Universal Robots PolyScope program: robot_interaction_lesson.urp

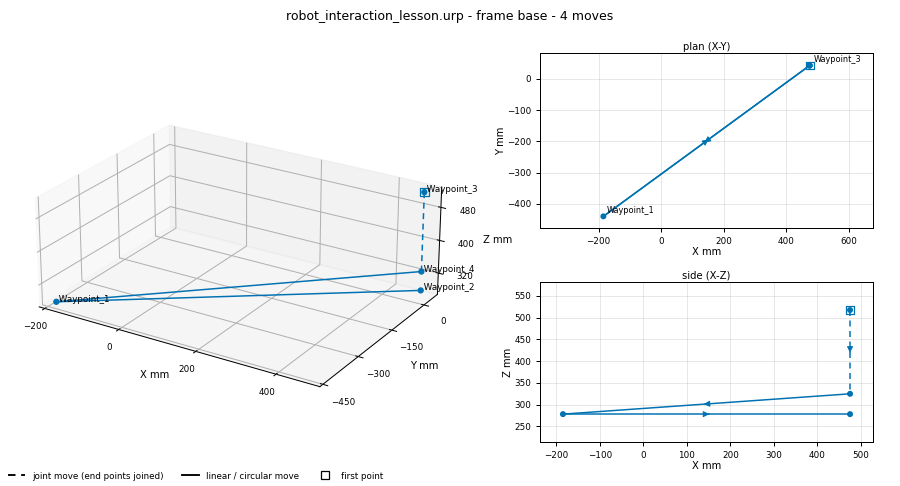
[picture p0: tool path of robot_interaction_lesson.urp in frame base, 4 of 4 moves have a stored position in this frame; points joined in program order, loops and branches not executed]
Program robot_interaction_lesson (installation=default directory=/ursim/programs createdIn=5.15.1 lastSavedIn=5.15.1 robotSerialNumber=20195699999)
Calibrated DH parameters: a=[0, -0.4784, -0.36, 0, 0, 0]; d=[0.1807, 0, 0, 0.17415, 0.11985, 0.11655]; alpha=[1.570796, 0, 0, 1.570796, -1.570796, 0]; deltaTheta=[0, 0, 0, 0, 0, 0]
InitVariablesNode variables(variable(name=returnVar, expression=0))
Robot Program (runOnlyOnce=true)
  Loop Forever
    Switch expression=returnVar
      Case (caseValue=1)
        Popup Message (haltProgram=false message=Wrist singularity inputType=Text)
        Loop Forever
          MoveJ speed 60 deg/s, acceleration 80 deg/s^2 (useActiveTCP=true) feature=Base
            Waypoint Waypoint_3: TCP in base x=474.982 y=42.583 z=517.603 mm, rx=2.6843 ry=-1.615 rz=-0.0538 rad; joints [26.177, -86.266, -97.066, -88.141, 91.393, -1.776] deg
            Waypoint Waypoint_4: TCP in base x=474.982 y=42.583 z=325.061 mm, rx=2.6843 ry=-1.615 rz=-0.0538 rad; joints [26.177, -94.555, -121.715, -55.204, 91.393, -1.776] deg
        returnVar := 0
      Case (caseValue=2)
        Popup Message (haltProgram=false message=Elbow singularity inputType=Text)
        MoveL speed 250 mm/s, acceleration 1200 mm/s^2 (useActiveTCP=true) feature=Base
          Waypoint Waypoint_1: TCP in base x=-184.548 y=-439.731 z=278.361 mm, rx=-0.0012 ry=3.1163 rz=0.0389 rad; joints [-91.713, -98.956, -126.223, -46.295, 91.392, -1.776] deg
          Waypoint Waypoint_2: TCP in base x=474.982 y=42.583 z=278.361 mm, rx=2.6843 ry=-1.615 rz=-0.0538 rad; joints [26.177, -98.956, -126.223, -46.295, 91.392, -1.776] deg; TCP offset x=0 y=0 z=0 mm, rx=0 ry=0 rz=0 rad
        returnVar := 0
      Case (caseValue=2147483647)
        Popup Message (haltProgram=false message=<html>Wrist singularity=1<br>Elbow singularity=2<br>Pick up tool=3</html> inputType=Text)
        Script: returnVar = request_integer_from_primary_client(">Wrist=1, Elbow=2 PnP=3")
